FUNCTION_BLOCK FB_1s_UPS_Base IMPLEMENTS I_1s_UPS
VAR
	_PcAmsNetId				:AMSNETID;			//PC AMS Net ID	
	
	_bReady					:BOOL;				//電源供給あり
	_e1sUpsState			:E_S_UPS_State;		//1s UPSのステータス
	
	{attribute 'TcPersistent'}
	_bPowerFailDetect		:BOOL;				//停電検知記憶
END_VAR

METHOD AcknowledgePowerFailDetect
_bPowerFailDetect:=FALSE;
END_METHOD

PROPERTY bPowerFailDetect : BOOL
GET
bPowerFailDetect:=_bPowerFailDetect;
END_GET
END_PROPERTY

PROPERTY bReady : BOOL
GET
bReady:=_bReady;
END_GET
END_PROPERTY

PROPERTY e1sUpsState : E_S_UPS_State
GET
e1sUpsState:=_e1sUpsState;
END_GET
END_PROPERTY

METHOD Execute
END_METHOD

//FB_Init は常に暗黙的に使用可能で、主に初期化に使用されます。
//戻り値は評価されません。特定の結果を得るために、メソッドを明示的に宣言し、
//そのメソッドに標準の初期化コードをもったコードを追加することができます。戻り値を評価できます。
METHOD FB_Init: BOOL
VAR_INPUT
    bInitRetains: BOOL; // TRUE: 保持変数は初期化されます (ウォーム リセット、あるいはコールド リセット)
    bInCopyCode: BOOL;  // TRUE: 後でコードをコピーする (オンライン変更) ために、インスタンスをコピーします。

	PcAmsNetId					:AMSNETID;		//PC AMS Net ID
END_VAR
_PcAmsNetId:=PcAmsNetId;
END_METHOD

END_FUNCTION_BLOCK

(* stored: Version 1.1.0.1
   POU FB_1s_UPS_Base: Id {d307deb9-28d5-4c30-a4c8-246804a0b876}, SpecialFunc None
   Method AcknowledgePowerFailDetect: Id {856d4f3b-c5ca-47e3-b4a8-32687b24ac83}
   Property bPowerFailDetect: Id {71da8cbe-9842-47a2-b993-f0955e0350af}
   Get Get: Id {a0dc9dff-8cbd-47a0-8567-b0e57c85eec9}
   Property bReady: Id {c9df24a0-69f7-4985-a7ed-3cf593322957}
   Get Get: Id {c195ff3a-f52c-47ac-848c-7b1555f6bd0f}
   Property e1sUpsState: Id {009aae78-1ffe-46fe-902a-191b0bf6d8ee}
   Get Get: Id {9fa6c78a-2452-448b-b165-39d017a0e4be}
   Method Execute: Id {9865cb07-5bf9-4cf4-87ed-c272c1d78e85}
   Method FB_Init: Id {ca250b63-edea-42e3-b08d-73d7a603dc14} *)
